// TIA Portal V20 export
DATA_BLOCK "PeaInformationLabel"   // DB14
TITLE = PeaInformationLabel
{ S7_Optimized_Access := 'TRUE' }
AUTHOR : Siemens AG
FAMILY : MTP
VERSION : 1.0
// List of product- and instance-specific information for the PEA handling within a modular plant environment.
// stored: DBAccessibleFromWebserver false, InstanceOfName typeMTPPeaInformationLabel, InstanceOfType UDT
"typeMTPPeaInformationLabel"
   // VAR
   //    AssetId : String := 'C1B54EEF-2D71-47BB-85AA-6F49015D382A';
   //    ComponentName : String := 'TesseractPEA';
   //    DeviceClass : String := 'ReactorService';
   //    DeviceHealth { ExternalWritable := 'False'} : Byte := 16#FF;
   //    DeviceManual { ExternalWritable := 'False'} : String := 'Reactor';
   //    DeviceRevision { ExternalWritable := 'False'} : String := '1.0.2';
   //    HardwareRevision { ExternalWritable := 'False'} : String := '1.0.2';
   //    Manufacturer { ExternalWritable := 'False'} : String := 'Siemens Presales Support';
   //    ManufacturerUri { ExternalWritable := 'False'} : String := 'https://support.industry.siemens.com/cs/de/de/view/109810699';
   //    Model { ExternalWritable := 'False'} : String := 'PresalesSupportExclusiveService';
   //    ProductCode { ExternalWritable := 'False'} : String := 'PresalesSupportPEA01';
   //    ProductInstanceUri { ExternalWritable := 'False'} : String := 'http://prtal.siemens.com/C1B54EEF-2D71-47BB-85AA-6F49015D382A';
   //    RevisionCounter { ExternalWritable := 'False'} : Int := 10;
   //    SerialNumber { ExternalWritable := 'False'} : String := 'C1B54EEF-2D71-47BB-85AA-6F49015D382A';
   //    SoftwareRevision { ExternalWritable := 'False'} : String := '2.8.0';
   // END_VAR
BEGIN
END_DATA_BLOCK
